Staubli VAL3: motionBuffer.pgx

public program motionBuffer(num x_nMovePts, num x_nElems)
begin

  // Do nothing
  // See start() program for more details

end
